// TwinCAT 3 PLC project PLC_SerialCom_Sample1
// ProgramVersion: 3.1.0.8
// libraries:
//   Tc2_SerialCom, * (Beckhoff Automation GmbH)
//   Tc2_Standard, * (Beckhoff Automation GmbH)
//   Tc3_Module, * (Beckhoff Automation GmbH)
// project tree:
//   GVLs/ GVL.TcGVL (not stored)
//   / PlcTask_Fast.TcTTO, PlcTask_Standard.TcTTO
//   POUs/ Background.TcPOU (not stored), BackgroundKL.TcPOU (not stored), BackgroundEL.TcPOU, FB_SerialCom.TcPOU (not stored), MAIN.TcPOU (not stored), BackgroundPcCOM.TcPOU
// real-time tasks:
//   TASK PlcTask_Fast: cycle T#2ms, priority 19, ADS port 350
//   TASK PlcTask_Standard: cycle T#10ms, priority 20, ADS port 351
// I/O:
//   DEVICE Device 3 (EtherCAT) (disabled), AmsNetId 172.17.60.154.4.1
//     Term 1 (EK1100) [EK1100 EtherCAT Coupler (2A E-Bus)]
//       Term 2 (EL6001) [EL6001 Interface (RS232)]
//       Box 3 (BK1250)
//   DEVICE Device 1 (NOV-DP-RAM)
//   DEVICE Device 2 (CX7000), AmsNetId 5.132.90.65.3.1
//     Term 2 (CX7028) [CX7028-0000-0118]
//       modules: Module 1 (DIO_2x), Module 3 (DIO_2x), Module 5 (DI_2x), Module 7 (DI_2x)
//   DEVICE Device 8 (COM Port)
// variable links:
//   PLC_SerialCom_Sample1/PLC_SerialCom_Sample1 Instance <-> Device 3 (EtherCAT)/Term 1 (EK1100)/Box 3 (BK1250)
//     PlcTask_Fast Inputs/BackgroundKL.stIn_KL6001/D[0] <-> Term 3 (KL6001-A)/Channel 1/Data In 0
//     PlcTask_Fast Inputs/BackgroundKL.stIn_KL6001/D[1] <-> Term 3 (KL6001-A)/Channel 1/Data In 1
//     PlcTask_Fast Inputs/BackgroundKL.stIn_KL6001/D[2] <-> Term 3 (KL6001-A)/Channel 1/Data In 2
//     PlcTask_Fast Inputs/BackgroundKL.stIn_KL6001/SerStatus <-> Term 3 (KL6001-A)/Channel 1/Ser. State
//     PlcTask_Fast Inputs/BackgroundKL.stIn_KL6001/Status <-> Term 3 (KL6001-A)/Channel 1/State
//     PlcTask_Fast Outputs/BackgroundKL.stOut_KL6001/Ctrl <-> Term 3 (KL6001-A)/Channel 1/Ctrl
//     PlcTask_Fast Outputs/BackgroundKL.stOut_KL6001/D[0] <-> Term 3 (KL6001-A)/Channel 1/Data Out 0
//     PlcTask_Fast Outputs/BackgroundKL.stOut_KL6001/D[1] <-> Term 3 (KL6001-A)/Channel 1/Data Out 1
//     PlcTask_Fast Outputs/BackgroundKL.stOut_KL6001/D[2] <-> Term 3 (KL6001-A)/Channel 1/Data Out 2
//     PlcTask_Fast Outputs/BackgroundKL.stOut_KL6001/SerCtrl <-> Term 3 (KL6001-A)/Channel 1/Ser. Ctrl
//   PLC_SerialCom_Sample1/PLC_SerialCom_Sample1 Instance <-> Device 3 (EtherCAT)/Term 1 (EK1100)/Term 2 (EL6001)
//     PlcTask_Fast Inputs/BackgroundEL.stIn_EL6001/D <-> Inputs/Data In 0
//     PlcTask_Fast Inputs/BackgroundEL.stIn_EL6001/D @bit {8..168 step 8} <-> Inputs/Data In {1..21}  (21 links)
//     PlcTask_Fast Inputs/BackgroundEL.stIn_EL6001/Status <-> Inputs/Status
//     PlcTask_Fast Outputs/BackgroundEL.stOut_EL6001/Ctrl <-> Outputs/Ctrl
//     PlcTask_Fast Outputs/BackgroundEL.stOut_EL6001/D <-> Outputs/Data Out 0
//     PlcTask_Fast Outputs/BackgroundEL.stOut_EL6001/D @bit {8..168 step 8} <-> Outputs/Data Out {1..21}  (21 links)
//   PLC_SerialCom_Sample1/PLC_SerialCom_Sample1 Instance <-> Device 8 (COM Port)
//     PlcTask_Standard Inputs/BackgroundPcCOM.stIn_PcCom/D <-> Inputs/Data1
//     PlcTask_Standard Inputs/BackgroundPcCOM.stIn_PcCom/D @bit {8..504 step 8} <-> Inputs/Data{2..64}  (63 links)
//     PlcTask_Standard Inputs/BackgroundPcCOM.stIn_PcCom/SerStatus <-> Inputs/Status
//     PlcTask_Standard Outputs/BackgroundPcCOM.stOut_PcCom/D <-> Outputs/Data1
//     PlcTask_Standard Outputs/BackgroundPcCOM.stOut_PcCom/D @bit {8..504 step 8} <-> Outputs/Data{2..64}  (63 links)
//     PlcTask_Standard Outputs/BackgroundPcCOM.stOut_PcCom/SerCtrl <-> Outputs/Ctrl

CONFIGURATION PLC_SerialCom_Sample1
    RESOURCE PLC ON TwinCAT3
        TASK PlcTask_Fast(INTERVAL := T#2ms, PRIORITY := 19);
        TASK PlcTask_Standard(INTERVAL := T#10ms, PRIORITY := 20);
        PROGRAM Background WITH PlcTask_Fast : Background;
        PROGRAM MAIN WITH PlcTask_Standard : MAIN;
    END_RESOURCE
END_CONFIGURATION

// ---- POUs/BackgroundEL.TcPOU
PROGRAM BackgroundEL
VAR
	(* background communication with the EL6001 terminal *)
	fbEL6001Ctrl		: SerialLineControl;
	bEL6001CtrlError	: BOOL;
	eEL6001CtrlErrorID	: ComError_t;
	(* 	I/O variables for a EL6001 terminal*)
	stIn_EL6001 AT %I*	: EL6inData22B;	(* linked to the EL6001 in the TwinCAT System Manager *)
	stOut_EL6001 AT %Q*	: EL6outData22B;(* linked to the EL6001 in the TwinCAT System Manager *)
END_VAR

(*
The SerialLineControl function block is supposed to be called in every PLC cycle.
It communicates with the serial line hardware device and transmits or receives data.
The SerialLineControl can be called in the standard task (e.g.for PcCOM port usage) 
or in a separate fast task (e.g.for terminal usage) as well.
A fast separate task will be necessary at high baud rates or with KL6001 terminals 
which have a small process image (3 or 5 data bytes only)
*)

(* background communication with the EL6001 terminal *)
fbEL6001Ctrl(
	Mode:= SERIALLINEMODE_EL6_22B, 
	pComIn:= ADR(stIn_EL6001), 
	pComOut:= ADR(stOut_EL6001), 
	SizeComIn:= SIZEOF(stIn_EL6001), 
	Error=> , 
	ErrorID=> , 
	TxBuffer:= TxBufferEL, 
	RxBuffer:= RxBufferEL );
IF fbEL6001Ctrl.Error THEN
	bEL6001CtrlError := TRUE;
	eEL6001CtrlErrorID := fbEL6001Ctrl.ErrorID;
END_IF

END_PROGRAM

// ---- POUs/BackgroundPcCOM.TcPOU
PROGRAM BackgroundPcCOM
VAR_IN_OUT
	RxBufferPcCom		: ComBuffer;	(* Receive data buffer; used with all receive function blocks *)
	TxBufferPcCom		: ComBuffer;	(* Transmit data buffer; used with all receive function blocks *)
END_VAR
VAR
	(* background communication with the PC COM port device *)
	fbPcComCtrl			: SerialLineControl;
	bPcComCtrlError		: BOOL;
	ePcComCtrlErrorID	: ComError_t;	
	(* 	I/O variables for a PC-COM port *)
	stIn_PcCom AT %I*	: PcComInData;	(* linked to the port in the TwinCAT System Manager *)
	stOut_PcCom AT %Q*	: PcComOutData;	(* linked to the port in the TwinCAT System Manager *)
END_VAR

(*
The SerialLineControl function block is supposed to be called in every PLC cycle.
It communicates with the serial line hardware device and transmits or receives data.
The SerialLineControl can be called in the standard task (e.g.for PcCOM port usage) 
or in a separate fast task (e.g.for terminal usage) as well.
A fast separate task will be necessary at high baud rates or with KL6001 terminals 
which have a small process image (3 or 5 data bytes only)
*)

(* background communication with the PC COM port device *)
fbPcComCtrl(
	Mode:= SERIALLINEMODE_PC_COM_PORT, 
	pComIn:= ADR(stIn_PcCom), 
	pComOut:= ADR(stOut_PcCom), 
	SizeComIn:= SIZEOF(stIn_PcCom), 
	Error=> , 
	ErrorID=> , 
	TxBuffer:= TxBufferPcCom, 
	RxBuffer:= RxBufferPcCom );
IF fbPcComCtrl.Error THEN
	bPcComCtrlError := TRUE;
	ePcComCtrlErrorID := fbPcComCtrl.ErrorID;
END_IF

END_PROGRAM
